// Mitsubishi GX Works2 project: Tapping1   PLC: FX3U/FX3UC

// global labels: Global1
VAR_GLOBAL
  XXFeed AT D52 : INT;
  XXRun AT M51 : BOOL;
  XXTarget AT D51 : INT;
  XXCurrent AT D50 : INT;
  XXArray AT D53 : ARRAY [0..5] OF INT;
  Foil3 AT M20 : BOOL;
  Foil4 AT M21 : BOOL;
  XXIMin AT X000 : BOOL;
  ZZIMin AT X001 : BOOL;
  ZZIMax AT X002 : BOOL;
  FoilExtractorIMax AT X003 : BOOL;
  XXODirection AT Y004 : BOOL;
  XXOPulse AT Y000 : BOOL;
  ReadWrite485OToggle AT Y001 : BOOL;
  ZZOToggle AT Y002 : BOOL;
  FoilExtractorOToggle AT Y003 : BOOL;
  FoilBlockerOToggle AT Y005 : BOOL;
  ZZRun AT M53 : BOOL;
  ZZDirection AT M52 : BOOL;
  RunStop AT M24 : BOOL;
  RunTest AT M23 : BOOL;
  FoilBlocker AT M54 : BOOL;
  FoilExtractor AT M55 : BOOL;
  RunState AT D20 : INT;
  Run AT M22 : BOOL;
  XXCurrentPulse AT D8132 : DINT;
  Foil3Array AT D200 : ARRAY [0..5] OF INT;
  Foil4Array AT D206 : ARRAY [0..5] OF INT;
  Read485 AT M100 : BOOL;
  Write485 AT M110 : BOOL;
  FoilIndex AT D60 : INT;
  Read485Value AT D102 : INT;
  Write485Value AT D112 : INT;
  RunIsTest AT M25 : BOOL;
  XXDirection AT M50 : BOOL;
  RunFeedXX AT D21 : INT;
  TestSensorFoil AT M30 : BOOL;
  FoilExtractorMin AT M31 : BOOL;
  FoilExtractorMax AT M32 : BOOL;
  FoilBlockerMin AT M33 : BOOL;
  FoilBlockerMax AT M34 : BOOL;
  RunStopEmergency AT M26 : BOOL;
  TestSensorRequire AT D22 : INT;
  TestFoilTimeSeconds AT D23 : INT;
  MachineReady AT M27 : BOOL;
  Foil1Manual AT M28 : BOOL;
  Foil1ManualIRun AT X004 : BOOL;
END_VAR

// task Task_01 (event TRUE, interval 0, priority 31): POU_01

PROGRAM POU_01
VAR
  fRising : BOOL;
  fFalling : BOOL;
  fXXFeedPulse : INT;
  fFoilIndexLast : INT;
  fFoilChanged : BOOL;
  fTemp : BOOL;
  fArrayIndex : INT;
  fArrayIndexDouble : INT;
  fRunStart : BOOL;
  fArrayCount : INT;
END_VAR
VAR CONSTANT
  fFoil3Offset : INT := 170;
  fFoil4Offset : INT := 170;
END_VAR
VAR
  fXXTarR : BOOL;
  fZZCheck : BOOL;
  fZZReady : BOOL;
END_VAR
VAR CONSTANT
  fRead485ValueError : INT := 10;
END_VAR
VAR
  fRW485Skip : INT;
  fRW485Sample : INT;
  fRead485Done : BOOL;
  fGetOriginDone : BOOL;
  fWrite485Done : BOOL;
  fXXReady : BOOL;
  fStepReady : BOOL;
  fGetOrigin : BOOL;
  fZZTarR : BOOL;
  fFoilDone : BOOL;
  fFoilTimerEN : BOOL;
  fFoilExtractorTimerEN : BOOL;
END_VAR
VAR CONSTANT
  fFoil1ManualPosition : INT := 11000;
END_VAR
(*////////////////////////////////////////*)
(*  _____       _ _   _       _ _         *)
(* |_   _|     (_) | (_)     | (_)        *)
(*   | |  _ __  _| |_ _  __ _| |_ _______ *)
(*   | | | '_ \| | __| |/ _` | | |_  / _ \*)
(*  _| |_| | | | | |_| | (_| | | |/ /  __/*)
(* |_____|_| |_|_|\__|_|\__,_|_|_/___\___|*)
(*                                        *)
(*////////////////////////////////////////*)
MOV(M8002, H8087, D8120);
MOV(M8002, K20, D8129);
MOV(M8002, K0, D8121);
MOV(M8002, 200, D8145);
MOV(M8002, fFoil3Offset, Foil3Array[0]); MOV(M8002, fFoil3Offset + 3000, Foil3Array[1]); MOV(M8002, fFoil3Offset + 6000, Foil3Array[2]);
MOV(M8002, fFoil4Offset, Foil4Array[0]); MOV(M8002, fFoil4Offset + 2000, Foil4Array[1]); MOV(M8002, fFoil4Offset + 4000, Foil4Array[2]); MOV(M8002, fFoil4Offset + 6000, Foil4Array[3]);
MOV(M8002, 260, D100); MOV(M8002, 0, D101);
MOV(M8002, 262, D110); MOV(M8002, 0, D111);
MOV(M8002, 80, RunFeedXX);
RST(M8002, TestSensorFoil);
RST(M8002, MachineReady);
MOV(M8002, fRead485ValueError, Read485Value);
SET(NOT MachineReady, ReadWrite485OToggle);
OUT_T(NOT MachineReady, TC0, 80);
SET(NOT MachineReady AND (Read485Value = 0 OR Read485Value = 1), MachineReady);
SET(NOT MachineReady AND TC0 AND NOT fZZReady AND NOT fZZCheck, fZZCheck);
(*//////////////////////////////////*)
(*  _____   _____ _  _   ___  _____ *)
(* |  __ \ / ____| || | / _ \| ____|*)
(* | |__) | (___ | || || (_) | |__  *)
(* |  _  / \___ \|__   _> _ <|___ \ *)
(* | | \ \ ____) |  | || (_) |___) |*)
(* |_|  \_\_____/   |_| \___/|____/ *)
(*                                  *)
(*//////////////////////////////////*)                                  
(*IVWR(en, station: 262(4xxxx), parameter: 0(x0001), value: any, channel)*)
IVWR(M8122, D110, D111, Write485Value, K1); 
RST(M8029, Write485);
RST(M8121, Write485);
PLS(Write485, fRising); SET(fRising, M8122);
PLF(Write485, fFalling); SET(fFalling, fWrite485Done);
(**)
(*IVRD(en, station, parameter, channel, store device)*)
PLS(Read485, fRising); MOV(fRising, fRead485ValueError, Read485Value);
RST(M8123, M8123);
RST(M8121, Read485);
IVRD(Read485, D100, D101, K1, Read485Value);
RST(M8029, Read485);
(*////////////////////////////////////////////////////*)
(*  __  __       _                                    *)
(* |  \/  |     (_)                                   *)
(* | \  / | __ _ _ _ __    _ __ ___   ___ _ __  _   _ *)
(* | |\/| |/ _` | | '_ \  | '_ ` _ \ / _ \ '_ \| | | |*)
(* | |  | | (_| | | | | | | | | | | |  __/ | | | |_| |*)
(* |_|  |_|\__,_|_|_| |_| |_| |_| |_|\___|_| |_|\__,_|*)
(*                                                    *)
(*////////////////////////////////////////////////////*)
OUT(FoilIndex = 3, Foil3);
OUT(FoilIndex = 4, Foil4);
OUT(FoilIndex = 1, Foil1Manual);
SET(FoilIndex <> fFoilIndexLast, fFoilChanged);
SET(fFoilChanged AND RunState <> 0, fTemp); RST(fTemp, fFoilChanged); MOV(fTemp, fFoilIndexLast, FoilIndex); RST(fTemp, fTemp);
MOV(fFoilChanged, FoilIndex, fFoilIndexLast);
BMOV(Foil3 AND fFoilChanged, D200, K6, D53);
BMOV(Foil4 AND fFoilChanged, D206, K6, D53);
RST(fFoilChanged, fFoilChanged);
SET(RunState = 0, fTemp);
PLS(Run, fRising); MOV(fRising AND fTemp, 1, RunState); RST(fRising AND fTemp, RunIsTest); SET(fRising AND fTemp, fRunStart);
PLS(RunTest, fRising); MOV(fRising AND fTemp, 1, RunState); SET(fRising AND fTemp, RunIsTest); SET(fRising AND fTemp, fRunStart);
RST(fTemp, fTemp);
MOV(fRunStart AND MachineReady AND (Foil3 OR Foil4 OR Foil1Manual), 2, RunState);
MOV(fRunStart AND Foil3, 3, fArrayCount);
MOV(fRunStart AND Foil4, 4, fArrayCount);
RST(fRunStart, fArrayIndexDouble);
RST(fRunStart, fRunStart);
PLS(RunStopEmergency, fRising); SET(fRising, fTemp);
RST(fTemp, XXRun);
RST(fTemp, ZZRun);
RST(fTemp, RunState);
RST(fTemp, Read485);
RST(fTemp, Write485);
RST(fTemp, FoilExtractor);
RST(fTemp, FoilBlocker);
RST(fTemp, fZZCheck);
RST(fTemp, fXXTarR);
RST(fTemp, fZZTarR);
RST(fTemp, fTemp);
(*|||||||||||||||||||||||||||||||||||||||||||||||||||||||||||||||||||||||||||||||||||||||||||||||||||||||||||||||||||||||||||||||||||||||||||||||||||||||||||*)
(*|||||||||||||||||||||||||||||||||||||||||||||||||||||||||||||||||||||||||||||||||||||||||||||||||||||||||||||||||||||||||||||||||||||||||||||||||||||||||||*)
OUT(NOT M8147, fXXReady);
SET(fXXReady AND RunState = 2, fTemp);
SET(fTemp, fGetOrigin);
RST(fTemp, fGetOriginDone);
MOV(fTemp AND NOT ZZIMin, 10, RunState);
MOV(fTemp AND ZZIMin, 13, RunState);
RST(fTemp, fTemp);

OUT(fGetOrigin AND fXXReady, fStepReady);
(*/////////////////////////////////////////////////////*)
(*   _____      _                      _       _       *)
(*  / ____|    | |                    (_)     (_)      *)
(* | |  __  ___| |_   ____   ___  _ __ _  __ _ _ _ __  *)
(* | | |_ |/ _ \ __| |_  /  / _ \| '__| |/ _` | | '_ \ *)
(* | |__| |  __/ |_   / /  | (_) | |  | | (_| | | | | |*)
(*  \_____|\___|\__| /___|  \___/|_|  |_|\__, |_|_| |_|*)
(*                                        __/ |        *)
(*                                       |___/         *)
(*/////////////////////////////////////////////////////*)
(*Set direction*)
SET(fStepReady AND RunState = 10, fTemp); RST(fTemp, fZZTarR);
SET(fTemp, ReadWrite485OToggle);
RST(fTemp AND ZZDirection, ZZDirection);
RST(fTemp, fZZReady);
SET(fTemp, fZZCheck);
MOV(fTemp, 11, RunState); RST(fTemp, fTemp);
(*Run*)
SET(fStepReady AND RunState = 11 AND fZZReady, fTemp);
SET(fTemp, ZZRun);
MOV(fTemp, 12, RunState); RST(fTemp, fTemp);
(*Done*)
SET(fStepReady AND RunState = 12 AND fZZTarR, fTemp); RST(fTemp, fZZTarR);
RST(fTemp, ReadWrite485OToggle);
MOV(fTemp, 13, RunState); RST(fTemp, fTemp);
(*|||||||||||||||||||||||||||||||||||||||||||||||||||||||||||||||||||||||||||||||||||||||||||||||||||||||||||||||||||||||||||||||||||||||||||||||||||||||||||*)
(*|||||||||||||||||||||||||||||||||||||||||||||||||||||||||||||||||||||||||||||||||||||||||||||||||||||||||||||||||||||||||||||||||||||||||||||||||||||||||||*)
(*Get z origin -> Get x origin*)
SET(fStepReady AND RunState = 13, fTemp);
MOV(fTemp, 20, RunState); RST(fTemp, fTemp);
(*//////////////////////////////////////////////////////*)
(*   _____      _                       _       _       *)
(*  / ____|    | |                     (_)     (_)      *)
(* | |  __  ___| |_  __  __   ___  _ __ _  __ _ _ _ __  *)
(* | | |_ |/ _ \ __| \ \/ /  / _ \| '__| |/ _` | | '_ \ *)
(* | |__| |  __/ |_   >  <  | (_) | |  | | (_| | | | | |*)
(*  \_____|\___|\__| /_/\_\  \___/|_|  |_|\__, |_|_| |_|*)
(*                                         __/ |        *)
(*                                        |___/         *)
(*//////////////////////////////////////////////////////*)
(*Move back*)
SET(fStepReady AND RunState = 20, fTemp);
RST(fTemp, XXCurrentPulse); MOV(fTemp, -20000, XXTarget); MOV(fTemp, 10, XXFeed); SET(fTemp, XXRun);
MOV(fTemp, 21, RunState); RST(fTemp, fTemp);
(*Move forward*)
SET(fStepReady AND RunState = 21 AND fXXTarR, fTemp); RST(fTemp, fXXTarR);
MOV(fTemp, 2000, XXTarget); MOV(fTemp, 1, XXFeed); SET(fTemp, XXRun);
MOV(fTemp, 22, RunState); RST(fTemp, fTemp);
(*Stop when out*)
SET(fGetOrigin AND RunState = 22 AND NOT XXIMin, fTemp);
RST(fTemp, XXRun);
MOV(fTemp, 23, RunState); RST(fTemp, fTemp);
(*Move forward 3mm*)
SET(fStepReady AND RunState = 23 AND fXXTarR, fTemp); RST(fTemp, fXXTarR);
RST(fTemp, XXCurrentPulse); MOV(fTemp, 100, XXTarget); MOV(fTemp, 1, XXFeed); SET(fTemp, XXRun);
MOV(fTemp, 24, RunState); RST(fTemp, fTemp);
(*Done*)
SET(fStepReady AND RunState = 24 AND fXXTarR, fTemp); RST(fTemp, fXXTarR);
RST(fTemp, XXCurrentPulse); RST(fTemp, XXTarget); MOV(fTemp, RunFeedXX, XXFeed);
MOV(fTemp AND NOT Foil1Manual, 25, RunState);
MOV(fTemp AND Foil1Manual, 50, RunState);
RST(fTemp AND Foil1Manual, fGetOrigin);
SET(fTemp AND Foil1Manual, fGetOriginDone);
RST(fTemp, fTemp);
(*/////////////////////////////////////////////////////*)
(*  _____                                  __      _ _ *)
(* |  __ \                                / _|    (_) |*)
(* | |__) | __ ___ _ __   __ _ _ __ ___  | |_ ___  _| |*)
(* |  ___/ '__/ _ \ '_ \ / _` | '__/ _ \ |  _/ _ \| | |*)
(* | |   | | |  __/ |_) | (_| | | |  __/ | || (_) | | |*)
(* |_|   |_|  \___| .__/ \__,_|_|  \___| |_| \___/|_|_|*)
(*                | |                                  *)
(*                |_|                                  *)
(*/////////////////////////////////////////////////////*)
(*Set initial position*)
SET(fStepReady AND RunState = 25, fTemp);
RST(fTemp, FoilExtractor); SET(fTemp, FoilExtractorMin);
SET(fTemp, FoilBlocker);
MOV(fTemp, 14, TestSensorRequire);
MOV(fTemp, 26, RunState); RST(fTemp, fTemp);
(*Wait until meet*)
SET(fStepReady AND RunState = 26 AND FoilExtractorMin AND FoilBlockerMax, fTemp);
RST(fTemp, fGetOrigin);
SET(fTemp, fGetOriginDone);
MOV(fTemp, 27, RunState); RST(fTemp, fTemp);
(*|||||||||||||||||||||||||||||||||||||||||||||||||||||||||||||||||||||||||||||||||||||||||||||||||||||||||||||||||||||||||||||||||||||||||||||||||||||||||||*)
(*|||||||||||||||||||||||||||||||||||||||||||||||||||||||||||||||||||||||||||||||||||||||||||||||||||||||||||||||||||||||||||||||||||||||||||||||||||||||||||*)
(*Prepair foil -> Loop*);
OUT(fGetOriginDone AND fXXReady AND NOT RunStop, fStepReady);
SET(fStepReady AND RunState = 27, fTemp);
MOV(fTemp, 30, RunState); RST(fTemp, fTemp);
(*//////////////////////////*)
(*  _                       *)
(* | |                      *)
(* | |     ___   ___  _ __  *)
(* | |    / _ \ / _ \| '_ \ *)
(* | |___| (_) | (_) | |_) |*)
(* |______\___/ \___/| .__/ *)
(*                   | |    *)
(*                   |_|    *)
(*//////////////////////////*)
(*Get next x position*)
SET(fStepReady AND RunState = 30, fTemp);
SET(fTemp, fFoilTimerEN);
OUT_T(fFoilTimerEN, TC184, 10000);
MOV(fTemp, fArrayIndexDouble MOD fArrayCount, fArrayIndex);
MOV(fTemp AND fArrayIndexDouble >= fArrayCount, fArrayCount - fArrayIndex - 1, fArrayIndex);
MOV(fTemp, XXArray[fArrayIndex], XXTarget);
INC(fTemp, fArrayIndexDouble);
RST(fTemp AND fArrayIndexDouble = fArrayCount * 2, fArrayIndexDouble);
MOV(fTemp, 31, RunState); RST(fTemp, fTemp);
(*Move x*)
SET(fStepReady AND RunState = 31, fTemp);
SET(fTemp, XXRun);
MOV(fTemp, 32, RunState); RST(fTemp, fTemp);
(*Reached x -> Set z direction down*)
SET(fStepReady AND RunState = 32 AND fXXTarR, fTemp); RST(fTemp, fXXTarR);
SET(fTemp, ReadWrite485OToggle);
SET(fTemp AND NOT ZZDirection, ZZDirection);
RST(fTemp, fZZReady);
SET(fTemp, fZZCheck);
MOV(fTemp, 33, RunState); RST(fTemp, fTemp);
(*Run z down*)
SET(fStepReady AND RunState = 33 AND fZZReady, fTemp);
SET(fTemp, ZZRun);
MOV(fTemp, 34, RunState); RST(fTemp, fTemp);
(*Set z direction up*)
SET(fStepReady AND RunState = 34 AND fZZTarR, fTemp); RST(fTemp, fZZTarR);
SET(fTemp, ReadWrite485OToggle);
RST(fTemp AND ZZDirection, ZZDirection);
RST(fTemp, fZZReady);
SET(fTemp, fZZCheck);
MOV(fTemp, 35, RunState); RST(fTemp, fTemp);
(*Run z up*)
SET(fStepReady AND RunState = 35 AND fZZReady, fTemp);
SET(fTemp, ZZRun);
MOV(fTemp, 36, RunState); RST(fTemp, fTemp);
(*Run z done*)
SET(fStepReady AND RunState = 36 AND fZZTarR, fTemp); RST(fTemp, fZZTarR);
RST(fTemp, ReadWrite485OToggle);
RST(fTemp, fFoilDone);
SET(fTemp AND (fArrayIndexDouble = 0 OR fArrayIndexDouble = fArrayCount), fFoilDone);
MOV(fFoilDone, T184, TestFoilTimeSeconds);
RST(fFoilDone, fFoilTimerEN);
RST(fFoilDone, T184);
MOV(fTemp AND NOT fFoilDone, 30, RunState);
MOV(fTemp AND fFoilDone, 37, RunState);
RST(fTemp, fFoilDone);
RST(fTemp, fTemp);
(*Blocker down*)
SET(fStepReady AND RunState = 37, fTemp);
RST(fTemp, FoilBlocker);
MOV(fTemp, 3, TestSensorRequire);
MOV(fTemp, 38, RunState); RST(fTemp, fTemp);
(*Blocker down done -> extractor forward*)
SET(fStepReady AND RunState = 38 AND FoilBlockerMin, fTemp);
SET(fTemp, FoilExtractor);
MOV(fTemp, 2, TestSensorRequire);
MOV(fTemp, 39, RunState); RST(fTemp, fTemp);
(*Extractor forward done -> blocker up*)
SET(fStepReady AND RunState = 39 AND FoilExtractorMax, fTemp);
SET(fTemp, FoilBlocker);
MOV(fTemp, 4, TestSensorRequire);
MOV(fTemp, 40, RunState); RST(fTemp, fTemp);
(*Blocker up done -> extractor back*)
SET(fStepReady AND RunState = 40 AND FoilBlockerMax, fTemp);
RST(fTemp, FoilExtractor);
MOV(fTemp, 1, TestSensorRequire);
MOV(fTemp, 41, RunState); RST(fTemp, fTemp);
(*Extractor back done -> return*)
SET(fStepReady AND RunState = 41 AND FoilExtractorMin, fTemp);
MOV(fTemp AND RunIsTest, 0, RunState);
MOV(fTemp AND NOT RunIsTest, 30, RunState);
RST(fTemp, fTemp);
(*///////////////////////////////////*)
(*  __  __                         _ *)
(* |  \/  |                       | |*)
(* | \  / | __ _ _ __  _   _  __ _| |*)
(* | |\/| |/ _` | '_ \| | | |/ _` | |*)
(* | |  | | (_| | | | | |_| | (_| | |*)
(* |_|  |_|\__,_|_| |_|\__,_|\__,_|_|*)
(*                                   *)
(*///////////////////////////////////*)
(*Get static x position*)
SET(fStepReady AND RunState = 50, fTemp);
RST(fTemp, FoilExtractor);
RST(fTemp, FoilBlocker);
MOV(fTemp, fFoil1ManualPosition, XXTarget);
MOV(fTemp, 51, RunState); RST(fTemp, fTemp);
(*Dirty skip*)
Set(fStepReady AND RunState >= 50 AND RunState < 61, fTemp);
INC(fTemp, RunState); RST(fTemp, fTemp);
(*Move x*)
SET(fStepReady AND RunState = 61, fTemp);
SET(fTemp, XXRun);
MOV(fTemp, 62, RunState); RST(fTemp, fTemp);
(*Reached x -> Set z direction down*)
PLS(Foil1ManualIRun, fRising);
SET(fStepReady AND RunState = 62 AND fXXTarR AND fRising, fTemp);
SET(fTemp, ReadWrite485OToggle);
SET(fTemp AND NOT ZZDirection, ZZDirection);
RST(fTemp, fZZReady);
SET(fTemp, fZZCheck);
MOV(fTemp, 63, RunState); RST(fTemp, fTemp);
(*Run z down*)
SET(fStepReady AND RunState = 63 AND fZZReady, fTemp);
SET(fTemp, ZZRun);
MOV(fTemp, 64, RunState); RST(fTemp, fTemp);
(*Set z direction up*)
SET(fStepReady AND RunState = 64 AND fZZTarR, fTemp); RST(fTemp, fZZTarR);
SET(fTemp, ReadWrite485OToggle);
RST(fTemp AND ZZDirection, ZZDirection);
RST(fTemp, fZZReady);
SET(fTemp, fZZCheck);
MOV(fTemp, 65, RunState); RST(fTemp, fTemp);
(*Run z up*)
SET(fStepReady AND RunState = 65 AND fZZReady, fTemp);
SET(fTemp, ZZRun);
MOV(fTemp, 66, RunState); RST(fTemp, fTemp);
(*Run z done*)
SET(fStepReady AND RunState = 66 AND fZZTarR, fTemp); RST(fTemp, fZZTarR);
RST(fTemp, ReadWrite485OToggle);
MOV(fTemp, 62, RunState); RST(fTemp, fTemp);
(*|||||||||||||||||||||||||||||||||||||||||||||||||||||||||||||||||||||||||||||||||||||||||||||||||||||||||||||||||||||||||||||||||||||||||||||||||||||||||||*)
(*|||||||||||||||||||||||||||||||||||||||||||||||||||||||||||||||||||||||||||||||||||||||||||||||||||||||||||||||||||||||||||||||||||||||||||||||||||||||||||*)

(**)
SET(XXRun AND XXTarget = DINT_TO_INT(XXCurrentPulse), fTemp);
SET(fTemp, fXXTarR);
RST(fTemp, XXRun); RST(fTemp, fTemp);
PLS(M8012, fRising); MOV(fRising, DINT_TO_INT(XXCurrentPulse), XXCurrent);
PLS(XXRun, fRising); MOV(fRising, XXFeed * 100, fXXFeedPulse); RST(fRising, ZZRun);
DRVA(XXRun, XXTarget, fXXFeedPulse, XXOPulse, XXODirection);
RST(M8029, XXRun);
PLF(XXRun, fFalling); SET(fFalling, fXXTarR);
OUT(XXODirection, XXDirection);
RST(NOT XXDirection AND XXIMin, XXRun);
(**)

(**)
RST(ZZRun AND NOT fZZReady, ZZRun);
RST(Read485Value = 0 AND ZZIMax, ZZRun);
RST(Read485Value = 1 AND ZZIMin, ZZRun);
PLF(ZZRun, fFalling); SET(fFalling, fZZTarR);
PLS(ZZDirection, fRising); SET(fRising, fZZCheck);
PLF(ZZDirection, fFalling); SET(fFalling, fZZCheck);
(*|||||||||||||||||||||||||||||||||||||||||||||||||||||||||||||||||||||||||||||||||||||||||||||||||||||||||||||||||||||||||||||||||||||||||||||||||||||||||||*)
PLS(fZZCheck, fRising);
RST(fRising, ZZRun);
MOV(fRising AND ZZDirection, 0, Write485Value);
MOV(fRising AND NOT ZZDirection, 1, Write485Value);
RST(fRising, fZZReady);
RST(fRising, fRW485Skip);
RST(fRising, fRW485Sample);
RST(fRising, fWrite485Done);
INC(fZZCheck AND NOT fWrite485Done, fRW485Skip);
SET(fZZCheck AND NOT fWrite485Done AND fRW485Skip >= 100, Write485);
(*|||||||||||||||||||||||||||||||||||||||||||||||||||||||||||||||||||||||||||||||||||||||||||||||||||||||||||||||||||||||||||||||||||||||||||||||||||||||||||*)
INC(fZZCheck AND fWrite485Done, fRW485Skip);
SET(fZZCheck AND fWrite485Done AND fRW485Skip >= 100, Read485);
PLF(Read485, fFalling); SET(fFalling, fTemp);
RST(fTemp, fRW485Skip);
INC(fTemp, fRW485Sample);
SET(ZZDirection AND Read485Value = 0, fZZReady);
SET(NOT ZZDirection AND Read485Value = 1, fZZReady);
SET(fZZReady, fRead485Done);
SET(fTemp AND fRW485Sample = 20, fRead485Done);
RST(fRead485Done, fRW485Skip);
RST(fRead485Done, fRW485Sample);
RST(fRead485Done, fZZCheck);
RST(fRead485Done, fWrite485Done);
RST(fRead485Done, fRead485Done);
RST(fTemp, fTemp);
(**)

(**)
OUT(ZZRun, ZZOToggle);
OUT(FoilExtractor, FoilExtractorOToggle);
OUT(FoilBlocker, FoilBlockerOToggle);
(**)
PLS(FoilExtractorMin, fRising); RST(fRising, FoilExtractorMax);
PLS(FoilExtractorMax, fRising); RST(fRising, FoilExtractorMin);
PLS(FoilBlockerMin, fRising); RST(fRising, FoilBlockerMax);
PLS(FoilBlockerMax, fRising); RST(fRising, FoilBlockerMin);
(**)
PLS(FoilExtractorIMax, fRising); SET(fRising, fFoilExtractorTimerEN);
OUT_T(NOT FoilExtractor AND fFoilExtractorTimerEN, TC31, 5);
PLS(TC31, fRising); SET(fRising, FoilExtractorMin); RST(fRising, fFoilExtractorTimerEN);
SET(FoilExtractor AND fFoilExtractorTimerEN, FoilExtractorMax); RST(fRising, fFoilExtractorTimerEN);
OUT_T(NOT FoilBlocker, TC33, 3);
PLS(TC33, fRising); SET(fRising, FoilBlockerMin);
OUT_T(FoilBlocker, TC34, 3);
PLS(TC34, fRising); SET(fRising, FoilBlockerMax);
END_PROGRAM
